//add
FUNCTION_BLOCK FB_1
VAR_INPUT
	nIn1:		INT;
	nIn2:		INT;
END_VAR
VAR_OUTPUT
	nOut1:		INT;
END_VAR
VAR
END_VAR

nOut1:=nIn1+nIn2;

END_FUNCTION_BLOCK

(* stored: Version 1.1.0.1, ProductVersion 3.1.4024.3
   POU FB_1: Id {105f3ca5-a6d7-4d1f-994a-44dc5c5b136d}, SpecialFunc None *)
